KUKA KRL program: trabalho_concluido.src, trabalho_concluido.dat

--- trabalho_concluido.src ---
&ACCESS RV10
&REL 4
&PARAM TEMPLATE = C:\KRC\Roboter\Template\vorgabe
&PARAM EDITMASK = *
DEF trabalho_concluido( )
;FOLD PULSE 3333 'R4 trabalho concluido' State=TRUE Time=3 sec;%{PE}%R 8.2.24,%MKUKATPBASIS,%COUT,%VPULSE,%P 2:3333, 3:R4 trabalho concluido, 5:TRUE, 6:, 8:3
PULSE($OUT[3333], TRUE,3)
;ENDFOLD

END

--- trabalho_concluido.dat ---
&ACCESS RV10
&REL 4
&PARAM TEMPLATE = C:\KRC\Roboter\Template\vorgabe
&PARAM EDITMASK = *
DEFDAT trabalho_concluido
;FOLD EXTERNAL DECLARATIONS;%{PE}%V3.2.0,%MKUKATPBASIS,%CEXT,%VCOMMON,%P
;FOLD BAS EXT;%{PE}%V3.2.0,%MKUKATPBASIS,%CEXT,%VEXT,%P
EXT  BAS (BAS_COMMAND  :IN,REAL  :IN )
DECL INT SUCCESS
;ENDFOLD
;FOLD GRIPPER EXT;%{E}%V3.2.0,%MKUKATPGRIPPER,%CEXT,%VEXT,%P
EXT  H50 (INT:IN, INT:IN ,INT:IN ,GRP_TYP:IN)
;ENDFOLD
;FOLD SPOT EXT;%{E}%V3.2.0,%MKUKATPSPOT,%CEXT,%VEXT,%P
EXT  USERSPOT (S_COMMAND  :IN, SPOT_TYPE:IN)
;ENDFOLD
;FOLD USER EXT;%{E}%V3.2.0,%MKUKATPUSER,%CEXT,%VEXT,%P
;Make here your modifications
;ENDFOLD
;ENDFOLD

ENDDAT
